(* PLC project FBD_EVOLUTION_8, Beckhoff Automation GmbH TwinCAT PLC Control 3.5.10.30 *)
(* stored: creationDateTime 2019-09-26T17:10:18.8029406, modificationDateTime 2019-09-26T17:10:18.8029406 *)

PROGRAM POU
VAR
	A: BOOL;
	B: BOOL;
	C: BOOL;
	D: BOOL;
END_VAR

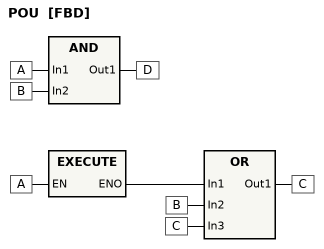
(* FBD diagram, written out as Structured Text *)
D := A AND B;
IF A THEN
  A := B AND C;
END_IF;
C := A OR B OR C;
END_PROGRAM

CONFIGURATION Application
  RESOURCE FBD_EVOLUTION_8 ON PLC
(* global variable list GVL *)
{attribute 'qualified_only'}
VAR_GLOBAL
	IsSFCResetting : BOOL;
END_VAR
    TASK PlcTask(INTERVAL := T#0ms, PRIORITY := 20);
    PROGRAM MAIN WITH PlcTask : MAIN;
  END_RESOURCE
END_CONFIGURATION
